(* CODESYS project A2HTC_VISU.project

Project tree, tasks and I/O mapping:
  Device : 750-8212 PFC200, WAGO, order no. 750-8212, version 6.3.0.12
    application Application
      libraries: Standard, 3.5.18.0 (System); CmpBitmapPool, * (System); VisuDialogs, * (System); Util, 3.5.21.0 (System); WagoSysModule_75x_640, 1.9.1.0 (WAGO); WagoAppTime, 1.7.3.5 (WAGO); SysTypes, * (System); SysTime, 3.5.17.0 (System); SysTimeRtc, * (System); CmpLog, * (System); CommFB, * (3S - Smart Software Solutions GmbH)
      task VISU_TASK (cyclic, interval 100 ms, priority 15) calls VisuElems.Visu_Prg, VisuSync
      task TrendRecordingTask (cyclic, interval 100 ms, priority 15) calls VisuTrendStorageAccess.GlobalInstances.g_TrendRecordingManager.CyclicCall
      task MainTask (cyclic, interval 200 ms, priority 15) calls PLC_PRG, readtest, TrendStorageAPI_TestProg
      visualisation Page
      Prog/
        function FctSetDefaultDataCurve [ST]
        program Prog [ST]
      visualisation Visualization_1
      text list TextList
      Trend Recording Manager
        Visualization_1_Trend1
        Visualization_1_Trend2
        Trend1
        Visualization_1_Trend3
      Overlap/
        function FctGetXYValues [ST]
        data type ENUM_CMD_PENDING
        program Overlap [ST]
      program PLC_PRG [ST]
      data type STATUS
      visualisation Visualization
      program VisuSync [ST]
      data type LIMITS
      visualisation Visualization_2
      function block VISU [ST]
      function LIMIT_CHECK [ST]
      data type UNIT
      image pool ImagePool
      global variables GVL
      data type GRAPH_AXIS
      function block READ_TRENDS [ST]
      function block FB_TrendConsumer [ST]: SetDestination, ErrorOccurred, ReadingDataCompleted, TimestampRead, ValueRead, VariableConfigurationRead
      function block FB_ReadTrend [ST]
      function DAY_TO_TIME [ST]
      function block CYCLE_TIME [ST]
      function T_PLC_MS [ST]
      program readtest [ST]
      program TrendStorageAPI_TestProg [ST]
      function block TrendStorageReaderConsumer [ST]: VariableConfigurationRead, ErrorOccurred, TimestampRead, ValueRead, ReadingDataCompleted, SetDestination
      function block TrendStorageWriterListener [ST]: DataWritten
      Visualizations/
        visualisation MinMaxTimestamps
        visualisation ReadValues
        visualisation NewDataWritten
    Kbus : Kbus, WAGO, version 2.1.0.1
        unmapped channels: K-BUS diagnostics
    Serial
      COM1 : COM1, WAGO, version 0.0.0.19
  libraries: VisuSymbols, 4.5.0.0 (System); WagoVisuIcons, 1.1.0.8 (WAGO); WagoVisuIconsMaterialDesign, 1.0.0.2 (WAGO)
  5ce3da45-db07-42e7-a21c-a00fff4ed8f6|C:\Users\MartinStark\Documents\A2HTC\VISU\Grün\Temp_Hum_OK.svg
  5ce3da45-db07-42e7-a21c-a00fff4ed8f6|C:\Users\MartinStark\Documents\A2HTC\VISU\Grün\Cooling_OK.svg
  5ce3da45-db07-42e7-a21c-a00fff4ed8f6|C:\Users\MartinStark\Documents\A2HTC\VISU\Rot\FAN_ERROR.svg
  5ce3da45-db07-42e7-a21c-a00fff4ed8f6|C:\Users\MartinStark\Documents\A2HTC\VISU\Gelb\Hum_WARN.svg
  5ce3da45-db07-42e7-a21c-a00fff4ed8f6|C:\Users\MartinStark\Documents\A2HTC\VISU\Rot\Heating_ERROR.svg
  5ce3da45-db07-42e7-a21c-a00fff4ed8f6|C:\Users\MartinStark\Documents\A2HTC\VISU\Grün\Heating_OK.svg
  5ce3da45-db07-42e7-a21c-a00fff4ed8f6|C:\Users\MartinStark\Documents\A2HTC\VISU\Gelb\Heating_WARN.svg
  5ce3da45-db07-42e7-a21c-a00fff4ed8f6|C:\Users\MartinStark\Documents\A2HTC\VISU\Gelb\FAN_WARN.svg
  5ce3da45-db07-42e7-a21c-a00fff4ed8f6|C:\Users\MartinStark\Documents\A2HTC\VISU\Gelb\Cooling_WARN.svg
  5ce3da45-db07-42e7-a21c-a00fff4ed8f6|C:\Users\MartinStark\Documents\A2HTC\VISU\Grün\FAN_OK.svg
  text list GlobalTextList
  5ce3da45-db07-42e7-a21c-a00fff4ed8f6|C:\Users\MartinStark\Documents\A2HTC\VISU\Rot\Cooling_ERROR.svg
  5ce3da45-db07-42e7-a21c-a00fff4ed8f6|C:\Users\MartinStark\Documents\A2HTC\VISU\Gelb\Temp_Hum_WARN.svg
  5ce3da45-db07-42e7-a21c-a00fff4ed8f6|C:\Users\MartinStark\Documents\A2HTC\VISU\Hintergrund.png
  5ce3da45-db07-42e7-a21c-a00fff4ed8f6|C:\Users\MartinStark\Documents\A2HTC\VISU\Rot\Temp_Hum_ERROR.svg
  5ce3da45-db07-42e7-a21c-a00fff4ed8f6|C:\Users\MartinStark\Documents\A2HTC\VISU\Rot\Hum_ERROR.svg
  5ce3da45-db07-42e7-a21c-a00fff4ed8f6|C:\Users\MartinStark\Documents\A2HTC\VISU\A2HTC.png
  5ce3da45-db07-42e7-a21c-a00fff4ed8f6|C:\Users\MartinStark\Documents\A2HTC\VISU\Grün\HUM_OK.svg
  5ce3da45-db07-42e7-a21c-a00fff4ed8f6|C:\Users\MartinStark\Documents\GitHub\PLS\Mirroring_Webvisu\graph\visu\Model_Viewer\model\Image_0.png
  5ce3da45-db07-42e7-a21c-a00fff4ed8f6|C:\Users\MartinStark\Documents\GitHub\PLS\Mirroring_Webvisu\graph\visu\Model_Viewer\model\Fox.bin
  5ce3da45-db07-42e7-a21c-a00fff4ed8f6|C:\Users\MartinStark\Documents\GitHub\PLS\Mirroring_Webvisu\graph\visu\Model_Viewer\model\Fox.gltf
  5ce3da45-db07-42e7-a21c-a00fff4ed8f6|C:\Users\MartinStark\Documents\GitHub\PLS\Mirroring_Webvisu\graph\visu\Model_Viewer\model\AlloySand2_bump_normalmap.png
  5ce3da45-db07-42e7-a21c-a00fff4ed8f6|C:\Users\MartinStark\Documents\GitHub\PLS\Mirroring_Webvisu\graph\visu\Model_Viewer\model\I5C3D083F677C41699172E93241A6F1D3basecolortexture.png
  5ce3da45-db07-42e7-a21c-a00fff4ed8f6|C:\Users\MartinStark\Documents\GitHub\PLS\Mirroring_Webvisu\graph\visu\Model_Viewer\model\ICA6ACE20800D44CEA1C27E63EFB994CEbasecolortexture.png
  5ce3da45-db07-42e7-a21c-a00fff4ed8f6|C:\Users\MartinStark\Documents\GitHub\PLS\Mirroring_Webvisu\graph\visu\Model_Viewer\model\MetalsOrnamentalMetalsAluminumBrushed_normalmap.png
  5ce3da45-db07-42e7-a21c-a00fff4ed8f6|C:\Users\MartinStark\Documents\A2HTC\VISU\Schriftarten Test\Bahnschrift Light.svg
  5ce3da45-db07-42e7-a21c-a00fff4ed8f6|C:\Users\MartinStark\Documents\A2HTC\VISU\Schriftarten Test\ISOCPEUR.svg
  5ce3da45-db07-42e7-a21c-a00fff4ed8f6|C:\Users\MartinStark\Documents\A2HTC\VISU\Schriftarten Test\Segoe UI Light.svg
  5ce3da45-db07-42e7-a21c-a00fff4ed8f6|C:\Users\MartinStark\Documents\A2HTC\VISU\Schriftarten Test\Yu Gothic UI Light.svg
  5ce3da45-db07-42e7-a21c-a00fff4ed8f6|C:\Users\MartinStark\Documents\A2HTC\VISU\Schriftarten Test\Arial Nova Light.svg
*)

// Device/Application/STATUS
TYPE STATUS :
STRUCT
	OK      : BOOL;
	WARNING : BOOL;
	ERROR   : BOOL;
END_STRUCT
END_TYPE

// Device/Application/LIMITS
TYPE LIMITS :
STRUCT
	UPPER_LIMIT : REAL := 25;
	LOWER_LIMIT : REAL := 22.5;
END_STRUCT
END_TYPE

// Device/Application/Overlap/ENUM_CMD_PENDING
{attribute 'qualified_only'}
{attribute 'strict'}
TYPE ENUM_CMD_PENDING :
(
	NO_CMD,         // no command pending
	UPDATE,         // Update pending
	CLEAN           // Clean pending
);
END_TYPE

// Device/Application/UNIT
TYPE UNIT :
STRUCT
	VALUE   : REAL := 23.5;
	STATUS  : STATUS;
	LIMITS  : LIMITS;
END_STRUCT
END_TYPE

// Device/Application/GRAPH_AXIS
TYPE GRAPH_AXIS :
STRUCT
	sLabel: STRING;
	aData: ARRAY[0..1000] OF REAL;
    diNumOfData : DINT;
	sBorderColor : STRING;
	xFill : BOOL;
END_STRUCT
END_TYPE

// Device/Application/GVL
{attribute 'qualified_only'}
VAR_GLOBAL
	TEMP_DEV_STATUS       : DWORD;
	HUM_DEV_STATUS        : DWORD;
	FAN_DEVICE_STATUS     : DWORD;
	HEATING_DEVICE_STATUS : DWORD;
	COOLING_DEVICE_STATUS : DWORD;
	
	TEMP       : UNIT;
	TEMP_LIMIT : LIMITS;
	HUM        : UNIT;
	HUM_LIMIT  :LIMITS;
	AIRFLOW    : UNIT;
	FAN        : UNIT;
	HEAT       : UNIT;
	COOLING    : UNIT;
	
	AIRFLOW_LIMIT : LIMITS;
	HEAT_POWER : REAL;
	COOL_POWER : REAL;
	just_true : BOOL := TRUE;
END_VAR

// Device/Application/VisuSync
PROGRAM VisuSync

VAR_INPUT
   udiCycleCounter : UDINT;
END_VAR

udiCycleCounter := udiCycleCounter +1;

END_PROGRAM

// Device/Application/PLC_PRG
PROGRAM PLC_PRG
VAR
	generator1 : GEN;
	iSignal1 : INT;
	rSignalToRecord1 : REAL;
	xRecord : BOOL;
	random_temp : REAL;
	random_hum  : REAL;
	always_true : BOOL:= TRUE;
    (* Define the struct variable *)
    myAxis : GRAPH_AXIS;
    
    (* Trigger variable to update data *)
    bUpdateChart : BOOL := FALSE;
    
    sInputLabels : STRING(1000); 
	
	first_cycle : BOOL:= FALSE;
	
	
	
	
	
	
	
    (* Function Block Instance *)
    fbTrendReader : FB_ReadTrend;
    
    (* Data Structure for the Chart *)
    stMyChartData : GRAPH_AXIS;
    sMyLabels : STRING(2000);
    
    (* Control Variables *)
    xReadTrigger : BOOL;
    xDone : BOOL;
    xBusy : BOOL;
    xError : BOOL;
    sErrorMessage : STRING;
    
    (* Parameters *)
    dtStartTime : DT;
    dtEndTime : DT;
    sTrendName : STRING := 'Trend1'; (* MUST match the Trend Recording name in Visualization Manager *)
    
    (* Helper to calc times *)
    tDuration : TIME := T#1H; (* Read last 1 hour *)
    // fbGetTime : GetLocalTime; (* Placeholder: Use system specific time FB *)
    dtNow : DT := DT#2024-01-01-10:00:00; 
    
	
	
    stChartData : GRAPH_AXIS;
    xInit : BOOL := TRUE;	
	
	fbCycleTime : CYCLE_TIME;
	
	
    dtNow2 : DT;
    sCurrentTime : STRING;
	
	

    Result : RTS_IEC_RESULT;

    ltodNow : LTIME_OF_DAY;
    ldatNow : LDATE;
	
    stUTC_DateAndTime : SysTimeRtc.SYSTIME;
    ldtNow : LDATE_AND_TIME;
    udiResult : RTS_IEC_RESULT;
	
	
	
	
END_VAR











IF random_temp > 40 THEN
	random_temp := 0;
ELSE 
	random_temp := random_temp + 2;
END_IF

IF random_hum > 80 THEN
	random_hum := 0;
ELSE 
	random_hum := random_hum + 1;
END_IF



generator1(MODE := GEN_MODE.SINE, BASE := TRUE, PERIOD := TIME#10S, AMPLITUDE := 500, OUT => iSignal1);
rSignalToRecord1 := INT_TO_REAL(iSignal1)/100 + 20; 
xRecord := rSignalToRecord1 >= 20;




(* Initialize only once or on demand *)
IF xInit THEN
    (* 1. Set Style Properties - Using fields from graph/db/GRAPH_AXIS.ST *)
    stChartData.sLabel := 'Fixed Values Demo';
    stChartData.sBorderColor := 'rgb(54, 162, 235)'; (* Blue *)
    stChartData.xFill := FALSE;

    (* 2. Set 10 Fixed Data Points *)
    stChartData.aData[0] := 10.0;
    stChartData.aData[1] := 20.0;
    stChartData.aData[2] := 15.5;
    stChartData.aData[3] := 25.0;
    stChartData.aData[4] := 30.0;
    stChartData.aData[5] := 10.0;
    stChartData.aData[6] := 5.0;
    stChartData.aData[7] := 12.0;
    stChartData.aData[8] := 18.0;
    stChartData.aData[9] := 22.0;
    
    (* Set the number of valid data points *)
    stChartData.diNumOfData := 10;
       
    xInit := FALSE;
END_IF

END_PROGRAM

// Device/Application/FB_ReadTrend
FUNCTION_BLOCK FB_ReadTrend
VAR_INPUT
	xExecute : BOOL;
    sTrendName : STRING; 
    tStartTime : DT;
    tEndTime : DT;
    iChannelIndex : INT := 0; 
END_VAR
VAR_OUTPUT
	sLabels : STRING(2000); 
    xDone : BOOL;
    xBusy : BOOL;
    xError : BOOL;
    sError : STRING;
END_VAR
VAR
	step : INT := 0;
    fbTrendReader : VisuTrendStorageAccess.TrendStorageReader;
    fbTrendConsumer : FB_TrendConsumer;
    
    liStart : LINT;
    liEnd : LINT;
    eResult : VisuTrendStorageAccess.ETrendStorageReaderErrors;
END_VAR
VAR_IN_OUT
    stChartData : GRAPH_AXIS;
END_VAR


CASE step OF
    0: (* Idle *)
        IF xExecute THEN
            xBusy := TRUE;
            xDone := FALSE;
            xError := FALSE;
            sError := '';
            
            // Set up Consumer
            fbTrendConsumer.SetDestination(ADR(stChartData), ADR(sLabels), tStartTime);
            
            // Initialize Reader
            fbTrendReader.Initialize(sTrendName); // User docu says Initialize exists. Assuming sTrendName arg.
            
            // Convert DT to LINT (Timestamp). DT is seconds. Trend usually ms.
            liStart := DT_TO_LINT(tStartTime) * 1000;
            liEnd := DT_TO_LINT(tEndTime) * 1000;
            
            step := 10;
        END_IF
        
    10: (* Start Read *)
        eResult := fbTrendReader.Read(
            liTimstampFrom := liStart,
            liTimstampTo := liEnd,
            itfTrendStorageReaderConsumer := fbTrendConsumer
        );
        
        IF eResult = VisuTrendStorageAccess.ETrendStorageReaderErrors.NoError THEN
             // Done immediately (unlikely for large data but possible)
             stChartData.sLabel := 'Trend Data';
             stChartData.sBorderColor := 'blue';
             stChartData.xFill := FALSE;
             step := 20;
        ELSIF eResult = VisuTrendStorageAccess.ETrendStorageReaderErrors.AdditionalReadCallRequired THEN
             step := 11; // Continue Reading
        ELSIF eResult = VisuTrendStorageAccess.ETrendStorageReaderErrors.NotInitialized THEN
             sError := 'Not Initialized';
             xError := TRUE;
             step := 99;
        ELSE
             sError := 'Read Error';
             xError := TRUE;
             step := 99;
        END_IF
        
    11: (* Continue Reading *)
        eResult := fbTrendReader.ContinueReading(
            liTimstampFrom := liStart,
            liTimstampTo := liEnd,
            itfTrendStorageReaderConsumer := fbTrendConsumer
        );

         IF eResult = VisuTrendStorageAccess.ETrendStorageReaderErrors.NoError THEN
             step := 20;
         ELSIF eResult = VisuTrendStorageAccess.ETrendStorageReaderErrors.AdditionalReadCallRequired THEN
             // Stay in step 11
         ELSE
             sError := 'Continue Error';
             xError := TRUE;
             step := 99;
         END_IF

    20: (* Done *)
        xDone := TRUE;
        xBusy := FALSE;
        IF NOT xExecute THEN
            step := 0;
        END_IF
        
    99: (* Error *)
        xBusy := FALSE;
        IF NOT xExecute THEN
            step := 0;
        END_IF
        
END_CASE

END_FUNCTION_BLOCK

// Device/Application/FB_TrendConsumer
FUNCTION_BLOCK FB_TrendConsumer IMPLEMENTS VisuTrendStorageAccess.ITrendStorageReaderConsumer
VAR_INPUT
	pChartData : POINTER TO GRAPH_AXIS;
    pLabelString : POINTER TO STRING(2000);
    tStart : DT;
END_VAR
VAR_OUTPUT
END_VAR
VAR
    pAxis : POINTER TO GRAPH_AXIS;
    pLabels : POINTER TO STRING(2000);
    sLabels : STRING(2000); // Internal build buffer
    iMaxLabels : INT := 20;
    tStartTime : DT;
    iCurrentRow : DINT;
    rCurrentVal : REAL;
    xFirst : BOOL := TRUE;
	
    // DEBUG
    debug_CountValueRead : DINT;
    debug_LastLiValue : LINT;
    debug_LastTimestamp : LINT;
    debug_CountTimestampRead : DINT;
    debug_LastTimestampIndex : DINT;
    
    pLReal : POINTER TO LREAL;
END_VAR

METHOD SetDestination
VAR_INPUT
	pChartData : POINTER TO GRAPH_AXIS;
    pLabelString : POINTER TO STRING(2000);
    tStart : DT;
END_VAR
    pAxis := pChartData;
    pLabels := pLabelString;
    tStartTime := tStart;
    
    // Reset
    IF pAxis <> 0 THEN
        pAxis^.diNumOfData := 0;
    END_IF
    IF pLabels <> 0 THEN
        pLabels^ := '[';
        sLabels := '[';
    END_IF
    xFirst := TRUE;
END_METHOD

(* Notification, that an error occurred.*)
METHOD ErrorOccurred
VAR_INPUT
	(* The error, that occurred*)
	eETrendStorageReaderErrors	: VisuTrendStorageAccess.ETrendStorageReaderErrors;
	(* Identifies the step, where the error occurred	*)
	eDuringWhichStep	: VisuTrendStorageAccess.ETrendStorageReaderStep;
END_VAR
END_METHOD

(* Notification, that reading the data (i.e. the values) has been completed.*)
METHOD ReadingDataCompleted
// Finalize labels
IF pLabels <> 0 THEN
	pLabels^ := CONCAT(pLabels^, ']');
END_IF
END_METHOD

(* Notification, that a timestamp from TblTrendData has been read and can be processed.*)
METHOD TimestampRead
VAR_INPUT
	(* A 0-based index of the row read from TblTrendData*)
	diWhichRow	: DINT;
	(* The absolute timestamp, that was read from TblTrendData*)
	liTimestamp	: LINT;


END_VAR
VAR
    sTempLabel : STRING(80);
    ldtCurrent : LDATE_AND_TIME;
    diIndex : DINT;
END_VAR
    // Convert timestamp (uS or mS? Usually uS or mS from Trend. LINT is usually ms or us)
    // Assuming MS since 1970? Or LTIME?
    // Standard Trend timestamps are µs (microseconds) usually.
    // DT is Seconds.
    
    // For label generation:
    // For label generation:
    IF pAxis <> 0 AND pLabels <> 0 THEN
        diIndex := pAxis^.diNumOfData; 
        
        // DEBUG
        debug_CountTimestampRead := debug_CountTimestampRead + 1;
        debug_LastTimestampIndex := diIndex; // Check what index TimestampRead sees
        
        IF diIndex < 100 AND (diIndex < iMaxLabels) THEN
             // ... logic ...
             
             // Convert to LDT (High Res) if liTimestamp is in ms (matches current_time logic)
             // current_time uses: TO_LDT(val * LTIME#1ms)
             ldtCurrent := TO_LDT(liTimestamp * LTIME#1ms);
             
             sTempLabel := LDT_TO_STRING(ldtCurrent);
             // Format: LDT#2025-02-07-13:15:15.369...
             // Take right 15 chars to get "15:15.369..." approx
             sTempLabel := RIGHT(sTempLabel, 15); 
             
             IF NOT xFirst THEN
                 pLabels^ := CONCAT(pLabels^, ', "');
             ELSE
                 pLabels^ := CONCAT(pLabels^, '"');
                 xFirst := FALSE;
             END_IF
             pLabels^ := CONCAT(pLabels^, sTempLabel);
             pLabels^ := CONCAT(pLabels^, '"');
        END_IF
    END_IF
END_METHOD

(* Notification, that a variable value from TblTrendData has been read and can be processed.*)
METHOD ValueRead
VAR_INPUT
	(* A 0-based index of the row read from TblTrendData.*)
	diWhichRow	: DINT;
	(* A 0-based index of the variable within all variables*)
	iWhichVariable	: INT;
	(* The value, that was read from TblTrendData*)
	liValue	: LINT;
	(* Indicates, whether NULL is stored in the trend storage*)
	xValueNULL	: BOOL;
END_VAR
VAR
    diIndex : DINT;
END_VAR
IF pAxis <> 0 THEN
	diIndex := pAxis^.diNumOfData;
	
	debug_CountValueRead := debug_CountValueRead + 1;
	debug_LastLiValue := liValue;
	
	IF diIndex <= 1000 THEN
		 // Debug: check raw value.
		 IF NOT xValueNULL THEN
			// Interpreting bits: liValue (LINT) holds the bits of LREAL (usually).
			// Or REAL? Standard Codesys Trend uses LREAL.
			// We point an LREAL pointer to the address of liValue to read it as float.
			// Then cast to REAL for the chart array.
			pLReal := ADR(liValue);
			pAxis^.aData[diIndex] := TO_REAL(pLReal^); 
		 ELSE
			pAxis^.aData[diIndex] := -9999.0; // Debug nulls
		 END_IF
		 
		 pAxis^.diNumOfData := pAxis^.diNumOfData + 1;
	END_IF
END_IF
END_METHOD

(* Notification, that the variable configuration was read and reading of data will start immediately.*)
METHOD VariableConfigurationRead
VAR_INPUT
	(* Points to an array of TrendStorageVariableDescription Variables,
 where the configuration of the variables has been stored. This array
 contains the description of the variables, whose data will be read*)
	paTrendStorageVariableDescription	: POINTER TO ARRAY [0..0] OF VisuTrendStorageAccess.TrendStorageVariableDescription;
	(* The effective size of the array above, i.e. the number of variables*)
	iCountVariables	: INT;
END_VAR
END_METHOD

END_FUNCTION_BLOCK

// Device/Application/CYCLE_TIME
FUNCTION_BLOCK CYCLE_TIME
VAR_INPUT
	RST : BOOL;
END_VAR
VAR_OUTPUT
	ct_min : TIME;
	ct_max : TIME;
	ct_last : TIME;
	systime : TIME;
	sysdays : INT;
	cycles : DWORD;
END_VAR
VAR
	last_cycle : TIME;
	tx: TIME;
	init: BOOL;
END_VAR


tx := DWORD_TO_TIME(T_PLC_MS()) - last_cycle;
IF rst THEN
	ct_min := t#10h;
	ct_max := t#0ms;
	cycles := 0;
ELSIF last_cycle > t#0s THEN
	IF tx < ct_min THEN ct_min := tx;
	ELSIF tx > ct_max THEN ct_max := tx;
	END_IF;
	ct_last := tx;
ELSIF ct_min = t#0s THEN
	ct_min := t#0s - t#1ms;
END_IF;
IF init THEN
	systime := systime + tx;
		IF systime >= t#1d THEN
			systime := systime - t#1d;
			sysdays := sysdays + 1;
		END_IF;
END_IF;
init := TRUE;
last_cycle := last_cycle + tx;
cycles := cycles + 1;

END_FUNCTION_BLOCK

// Device/Application/T_PLC_MS
FUNCTION T_PLC_MS : DWORD
VAR CONSTANT
	debug : BOOL := 0;
	N : INT := 0;
	offset : DWORD := 0;
END_VAR
VAR
	tx : TIME;
END_VAR


tx := TIME();
T_PLC_MS := TIME_TO_DWORD(Tx);

IF debug THEN
	T_PLC_MS := (SHL(T_PLC_MS,N) OR SHL(DWORD#1,N)-1) + OFFSET;
END_IF;

END_FUNCTION

// Device/Application/readtest
PROGRAM readtest
VAR
	i : INT;
	
	diVal2 : DINT := 1000;
	siVal3 : SINT;
	
	rVal	: REAL;
	rSin	: REAL;
END_VAR

// This program simulates the data, that is written to the trend storage

i := (i + 1) MOD 23;
siVal3 := siVal3 + 1;

IF siVal3 > 0 THEN
	diVal2 := diVal2 + 2;
	
	IF diVal2 > 1100 THEN
		diVal2 := 1000;
	END_IF
END_IF

rVal := rVal +0.05;
rSin := 5 * SIN(rVal);

END_PROGRAM

// Device/Application/TrendStorageAPI_TestProg
// Example program, that access the trend storage
PROGRAM TrendStorageAPI_TestProg
VAR
	xInitialized : BOOL;
	instTrendStorageReader 			: TrendStorageReader; 
	instTrendStorageWriterListener	: TrendStorageWriterListener;
	instTrendStorageReaderConsumer	: TrendStorageReaderConsumer;
	
	// Usecase 1:
	eError							: VisuTrendStorageAccess.ETrendStorageReaderErrors;
	liMinTimestamp					: LINT;
	liMaxTimestamp					: LINT;
	timeDateMin						: SYSTIMEDATE;
	uiMicrosecondsMin				: UINT;
	timeDateMax						: SYSTIMEDATE;
	uiMicrosecondsMax				: UINT;
	
	// Usecase 2:
	xDoReadTest2					: BOOL;
	eError2							: VisuTrendStorageAccess.ETrendStorageReaderErrors;
	liTimstampFrom2					: LINT;
	liTimstampTo2					: LINT;
	iLoopCounter					: INT;
	
	xStopContinueReading			: BOOL;

	xComputeTimestamps				: BOOL;
	xComputeDateTime				: BOOL;
	timeDateFrom2					: SYSTIMEDATE;
	uiMicrosecondsFrom2				: UINT;
	timeDateTo2						: SYSTIMEDATE;
	uiMicrosecondsTo2				: UINT;
	
	
	ChartOne : GRAPH_AXIS;
	sLabelOne : STRING(2000);
	
	    stUTC_DateAndTime : SYSTIME;

    Result : RTS_IEC_RESULT;

    ldtNow : LDATE_AND_TIME;
    ltodNow : LTIME_OF_DAY;
    ldatNow : LDATE;

    stUTC_Timestamp : SysTime;
    stLocal_TimeStamp : SysTime;
    stdNow : SysTimeDate;

    dtNow : DATE_AND_TIME;
    todNow : TIME_OF_DAY;
    datNow : DATE;   
    datToday : DATE; 	
END_VAR

// Required call to Initialize before any methods of the TrendStorageReader instance can be used
Result := SysTimeRtcHighResGet(stUTC_DateAndTime); // UlINT#1738934115369

ldtNow := TO_LDT(stUTC_DateAndTime * LTIME#1ms); // LDT#2025-2-7-13:15:15.369000000
ltodNow := TO_LTOD(ldtNow); // LTOD#13:15:15.369000000
ldatNow := TO_LDATE(ldtNow); // LD#2025-2-7


Result := SysTimeRtcHighResGet(stUTC_Timestamp); // ULINT#1528273494913
Result := SysTimeRtcConvertHighResToLocal(stUTC_Timestamp, stdNow);

Result := SysTimeRtcConvertDateToHighRes(stdNow, stLocal_TimeStamp); // ULINT#1528280694913

dtNow := TO_DT(stLocal_TimeStamp / 1000); // DT#2018-6-6-10:24:54
todNow := TO_TOD(stLocal_TimeStamp MOD TO_ULINT(T#1D)); // TOD#10:24:54.913
datToday := TO_DATE(dtNow); // D#2018-6-6


// Required call to Initialize before any methods of the TrendStorageReader instance can be used
IF NOT xInitialized THEN
	xInitialized := TRUE;
	instTrendStorageReader.Initialize(sPacketName := 'Trend1');
	// Usecase 3: Notification, if new data is available in the trend storage.
	// This optional call is necessary, if we want to be informed, if new data has been written
	// to the trend storage.
	instTrendStorageReader.AddTrendStorageWriterListener(instTrendStorageWriterListener);
END_IF

// Usecase 1: Determine the min/max timestamp range, for which data is available in the trend storage
eError := instTrendStorageReader.GetMinMaxTimestamps(
	liMinTimestamp			=> liMinTimestamp,
	liMaxTimestamp			=> liMaxTimestamp
);

// Comvert the timestamps in a human readable form
TrendStorageConvertFromTimestamp(liTimestamp := liMinTimestamp, timeDate => timeDateMin, uiMicroseconds => uiMicrosecondsMin);
TrendStorageConvertFromTimestamp(liTimestamp := liMaxTimestamp, timeDate => timeDateMax, uiMicroseconds => uiMicrosecondsMax);

// Usecase 2: Read values from the trend storage
// The data returned by the read process is truncated into small pieces. The 1st call is a call
// of method Read. In case of return code VisuTrendStorageAccess.ETrendStorageReaderErrors.AdditionalReadCallRequired
// additional calls are necessary, but calls to method ContinueReading.
IF eError2 = VisuTrendStorageAccess.ETrendStorageReaderErrors.AdditionalReadCallRequired THEN
	iLoopCounter := iLoopCounter + 1;
	VisuElems.Visu_Output_2('Call to ContinueReading ', INT_TO_STRING(iLoopCounter), 4);
	eError2 := instTrendStorageReader.ContinueReading(
		liTimstampFrom					:= liTimstampFrom2,
		liTimstampTo					:= liTimstampTo2,
		itfTrendStorageReaderConsumer	:= instTrendStorageReaderConsumer
	);
END_IF

IF xDoReadTest2 THEN
	xDoReadTest2 := FALSE;

	iLoopCounter := 0;
	instTrendStorageReaderConsumer.diTotalCountRows := 0;
	
	instTrendStorageReaderConsumer.SetDestination(pChartData := ADR(ChartOne), pLabelString := ADR(sLabelOne), tStart := dtNow);

	// Always read full range
    liTimstampFrom2 := liMinTimestamp;
    liTimstampTo2 := liMaxTimestamp;
	
	eError2 := instTrendStorageReader.Read(
		liTimstampFrom					:= liTimstampFrom2,
		liTimstampTo					:= liTimstampTo2,
		itfTrendStorageReaderConsumer	:= instTrendStorageReaderConsumer
	);
END_IF

// This helps us to abort a long running read call
IF xStopContinueReading THEN
	xStopContinueReading := FALSE;
	// This stops the reading
	eError2 := VisuTrendStorageAccess.ETrendStorageReaderErrors.NoError;
END_IF

IF xComputeTimestamps THEN
	xComputeTimestamps := FALSE;
	
	liTimstampFrom2 := TrendStorageConvertToTimestamp(timeDateFrom2, uiMicrosecondsFrom2);
	liTimstampTo2 := TrendStorageConvertToTimestamp(timeDateTo2, uiMicrosecondsTo2);
END_IF

IF xComputeDateTime THEN
	 xComputeDateTime := FALSE;
	 
	TrendStorageConvertFromTimestamp(liTimestamp := liTimstampFrom2, timeDate => timeDateFrom2, uiMicroseconds => uiMicrosecondsFrom2);
	TrendStorageConvertFromTimestamp(liTimestamp := liTimstampTo2, timeDate => timeDateTo2, uiMicroseconds => uiMicrosecondsTo2);
END_IF

END_PROGRAM

// Device/Application/TrendStorageWriterListener
// Example function block, that will be informed, if new data has been written to the
// trend storage. It simply stores the information, that is displayed in the visualization
// "ReadValues"
FUNCTION_BLOCK TrendStorageWriterListener IMPLEMENTS ITrendStorageWriterListener
VAR
	m_liFirstTimestamp	: LINT;
	m_liLastTimestamp	: LINT;
	m_iCountRows		: INT;
	
	m_timeDateMin		: SYSTIMEDATE;
	m_uiMicrosecondsMin	: UINT;
	m_timeDateMax		: SYSTIMEDATE;
	m_uiMicrosecondsMax	: UINT;
END_VAR

(* Notification, that data has been written to the trend storage*)
METHOD DataWritten
VAR_INPUT
	(* The first timestamp for which data was written to the trend storage*)
	liFirstTimestamp	: LINT;
	(* The last timestamp for which data was written to the trend storage*)
	liLastTimestamp	: LINT;
	(* The number of rows, that have been written to the trend storage*)
	iCountRows	: INT;
END_VAR
m_liFirstTimestamp := liFirstTimestamp;
m_liLastTimestamp := liLastTimestamp;
m_iCountRows := iCountRows;

// Comvert the timestamps in a human readable form
TrendStorageConvertFromTimestamp(liTimestamp := liFirstTimestamp, timeDate => m_timeDateMin, uiMicroseconds => m_uiMicrosecondsMin);
TrendStorageConvertFromTimestamp(liTimestamp := liLastTimestamp, timeDate => m_timeDateMax, uiMicroseconds => m_uiMicrosecondsMax);
END_METHOD

END_FUNCTION_BLOCK

// Device/Application/TrendStorageReaderConsumer
// This function block is a simple example implementation of the ITrendStorageReaderConsumer interface.
FUNCTION_BLOCK TrendStorageReaderConsumer IMPLEMENTS ITrendStorageReaderConsumer
VAR_INPUT
	// If this flag is TRUE an output like a csv export will be generated. Should be only
	// used, if not too much data is read from the trend storage
	xDetailedOutput						: BOOL;
	
	// This member is used to track the total number of rows, that have been read from the trend storage
	diTotalCountRows					: DINT;
END_VAR
VAR
	// This instance converts the values into a suitable representation, e.g. into a string
	m_instValueConverter				: TrendStorageReaderValueConverter;	

	// A line used to collect the data read from the trend storage
	m_sLine								: STRING(255);
	// Used to identify the rows
	m_diWhichRow						: DINT;
	
	m_diRowCounter						: DINT;
	// Used to track the minimum/maximum timestamp, that was read
	m_liTimestampMin					: LINT := 16#1FFFFFFFFFFFFFFF;
	m_liTimestampMax					: LINT := 0;
	
	
	pAxis : POINTER TO GRAPH_AXIS;
    pLabels : POINTER TO STRING(2000);
    sLabels : STRING(2000);
    tStartTime : DT;
    xFirst : BOOL;	
	

    
    rLastNonZeroValue : REAL;	
	
    // Deep Debugging
    liLastRawValue : LINT;
    iLastVarIndex : INT;
    diValueReadCalls : DINT;
    xLastNull : BOOL;	
END_VAR

METHOD VariableConfigurationRead
VAR_INPUT
	paTrendStorageVariableDescription	: POINTER TO ARRAY [0..0] OF VISUTRENDSTORAGEACCESS.TrendStorageVariableDescription;
	iCountVariables	: INT;
END_VAR
m_instValueConverter.SetVariableConfiguration(paTrendStorageVariableDescription, iCountVariables);

// If we previously collected data, we dump it
//ReadingDataCompleted();

VisuElems.Visu_Output_3('New configuration having ', INT_TO_STRING(iCountVariables), ' variables', 4);
END_METHOD

METHOD ErrorOccurred
VAR_INPUT
	(* The error, that occurred*)
	eETrendStorageReaderErrors	: VISUTRENDSTORAGEACCESS.ETrendStorageReaderErrors;
	(* Identifies the step, where the error occurred	*)
	eDuringWhichStep	: VISUTRENDSTORAGEACCESS.ETrendStorageReaderStep;
END_VAR
// Error processing can be done here...
END_METHOD

(* Notification, that a timestamp from TblTrendData has been read and can be processed.*)
METHOD TimestampRead
VAR_INPUT
	(* A 0-based index of the row read from TblTrendData*)
	diWhichRow	: DINT;
	
	(* The absolute timestamp, that was read from TblTrendData*)
	liTimestamp	: LINT;
END_VAR
VAR
	timeDate		: SYSTIMEDATE;
	uiMicroseconds	: UINT;
END_VAR

IF xDetailedOutput THEN
	IF LEN(m_sLine) <> 0 THEN
		VisuElems.Visu_Output_3(DINT_TO_STRING(m_diWhichRow), ': ', m_sLine, 4);
	END_IF
	m_sLine := '';
END_IF

m_diWhichRow := diWhichRow;


IF xDetailedOutput THEN
	// We begin a new line
	m_sLine := LINT_TO_STRING(liTimestamp);

	// Comvert the timestamps in a human readable form
	TrendStorageConvertFromTimestamp(liTimestamp := liTimestamp, timeDate => timeDate, uiMicroseconds => uiMicroseconds);

	// We also append the timestamp in the human readable way
	m_sLine := CONCAT(m_sLine, ';');
	m_sLine := CONCAT(m_sLine, WORD_TO_STRING(timeDate.wYear));
	m_sLine := CONCAT(m_sLine, '-');
	m_sLine := CONCAT(m_sLine, WORD_TO_STRING(timeDate.wMonth));
	m_sLine := CONCAT(m_sLine, '-');
	m_sLine := CONCAT(m_sLine, WORD_TO_STRING(timeDate.wDay));
	m_sLine := CONCAT(m_sLine, ' ');
	m_sLine := CONCAT(m_sLine, WORD_TO_STRING(timeDate.wHour));
	m_sLine := CONCAT(m_sLine, ':');
	m_sLine := CONCAT(m_sLine, WORD_TO_STRING(timeDate.wMinute));
	m_sLine := CONCAT(m_sLine, ':');
	m_sLine := CONCAT(m_sLine, WORD_TO_STRING(timeDate.wSecond));
	m_sLine := CONCAT(m_sLine, ':');
	m_sLine := CONCAT(m_sLine, WORD_TO_STRING(timeDate.wMilliseconds));
	m_sLine := CONCAT(m_sLine, ':');
	m_sLine := CONCAT(m_sLine, UINT_TO_STRING(uiMicroseconds));
ELSE
	m_diRowCounter := m_diRowCounter + 1;
	
	m_liTimestampMax := MAX(m_liTimestampMax, liTimestamp);
	
	(* Append to Label String - Protect against overflow *)
	IF pLabels <> 0 AND LEN(pLabels^) < 1900 THEN
	    TrendStorageConvertFromTimestamp(liTimestamp := liTimestamp, timeDate => timeDate, uiMicroseconds => uiMicroseconds);
	    
	    IF NOT xFirst THEN
	        pLabels^ := CONCAT(pLabels^, ','); // Add comma separator
	    END_IF
	    xFirst := FALSE; 
	    
	    pLabels^ := CONCAT(pLabels^, '"');
	    pLabels^ := CONCAT(pLabels^, WORD_TO_STRING(timeDate.wHour));
	    pLabels^ := CONCAT(pLabels^, ':');
	    pLabels^ := CONCAT(pLabels^, WORD_TO_STRING(timeDate.wMinute));
	    pLabels^ := CONCAT(pLabels^, ':');
	    pLabels^ := CONCAT(pLabels^, WORD_TO_STRING(timeDate.wSecond));
	    pLabels^ := CONCAT(pLabels^, '"');
	END_IF
END_IF
END_METHOD

METHOD ValueRead
VAR_INPUT
	(* A 0-based index of the row read from TblTrendData.*)
	diWhichRow	: DINT;
	(* A 0-based index of the variable within all variables*)
	iWhichVariable	: INT;
	(* The value, that was read from TblTrendData*)
	liValue	: LINT;
	(* Indicates, whether NULL is stored in the trend storage*)
	xValueNULL	: BOOL;
END_VAR
VAR
	sValue		: STRING;
END_VAR

// Debug Capture
diValueReadCalls := diValueReadCalls + 1;
liLastRawValue := liValue;
iLastVarIndex := iWhichVariable;
xLastNull := xValueNULL;

IF xDetailedOutput THEN
	// We simply append the value to the line, that simulates a line of a csv file
	m_sLine := CONCAT(m_sLine, ';');
	
	sValue := m_instValueConverter.ConvertToString(iWhichVariable, liValue, xValueNULL);
	m_sLine := CONCAT(m_sLine, sValue);
ELSE
    IF pAxis <> 0 THEN
        IF iWhichVariable = 0 AND NOT xValueNULL THEN
             IF pAxis^.diNumOfData <= 1000 THEN
                // Use converter to handle potential REAL/INT types correctly via string representation
                sValue := m_instValueConverter.ConvertToString(iWhichVariable, liValue, xValueNULL);
                pAxis^.aData[pAxis^.diNumOfData] := STRING_TO_REAL(sValue);
                
                IF pAxis^.aData[pAxis^.diNumOfData] <> 0 THEN
                    rLastNonZeroValue := pAxis^.aData[pAxis^.diNumOfData];
                END_IF
                
                pAxis^.diNumOfData := pAxis^.diNumOfData + 1;
            END_IF       
        END_IF
    END_IF

END_IF
END_METHOD

{attribute '''DOCU__COMMENT' := ' Notification, that reading the data (i.e. the values) has been completed.'}
(* Notification, that reading the data (i.e. the values) has been completed.*)
METHOD ReadingDataCompleted

VAR
	CMPID_LigLog: UDINT;
	sLogMessage : STRING(255);
END_VAR
IF xDetailedOutput THEN
	IF LEN(m_sLine) <> 0 THEN
		VisuElems.Visu_Output_3(DINT_TO_STRING(m_diWhichRow), ': ', m_sLine, 4);
	END_IF
	m_sLine := '';
ELSE
	diTotalCountRows := diTotalCountRows + m_diRowCounter;

	sLogMessage := CONCAT('ReadingDataCompleted, m_diRowCounter = ', CONCAT('ReadingDataCompleted, m_diRowCounter = ', CONCAT(', diTotalCountRows = ', DINT_TO_STRING(diTotalCountRows))));
	//LogAdd2(LOG_STD_LOGGER, 0, CmpLog.LogClass.LOG_INFO, 0, 0, sLogMessage);
	
	// Prepare for next loops
	m_diRowCounter := 0;
	m_liTimestampMin := 16#1FFFFFFFFFFFFFFF;
	m_liTimestampMax := 0;
	
	
	IF pLabels <> 0 THEN
	    pLabels^ := CONCAT(pLabels^, ']');
	END_IF	
END_IF
END_METHOD

METHOD SetDestination : BOOL
VAR_INPUT
    pChartData : POINTER TO GRAPH_AXIS;
    pLabelString : POINTER TO STRING(2000);
    tStart : DT;
END_VAR
    pAxis := pChartData;
    pLabels := pLabelString;
    tStartTime := tStart;
    
    // Reset
    IF pAxis <> 0 THEN
        pAxis^.diNumOfData := 0;
    END_IF
    IF pLabels <> 0 THEN
        pLabels^ := '[';
        sLabels := '[';
    END_IF
    xFirst := TRUE;
END_METHOD

END_FUNCTION_BLOCK

// Device/Application/Overlap/FctGetXYValues
/// Get X & Y values
FUNCTION FctGetXYValues : bool

VAR_INPUT
   iValue : INT;                     // Input value for calculation  
	rXValue : REFERENCE TO REAL;      // X value 
	rYValue : REFERENCE TO REAL;      // Y value 
END_VAR

VAR
   rValue : REAL;
END_VAR

// X = t − 2 sin t
// Y = 2 − 2 cos t

rValue  := INT_TO_REAL(iValue);
rValue  := rValue/10.0;
rXValue := rValue - 2.0*SIN(rValue);
rYValue := 2.0 - 2.0*COS(rValue);

END_FUNCTION

// Device/Application/Prog/FctSetDefaultDataCurve
/// Set default data for curves
FUNCTION FctSetDefaultDataCurve : bool

VAR
   ix : INT;
END_VAR

// Clean up the arrays
FOR ix := 1 TO 100 BY 1 DO
    Prog.DataX1[ix]  := 0.0 ;
    Prog.DataY1[ix]  := 0.0 ;
END_FOR
   
// Set deualt data   
Prog.DataX1[1] := -10.0 ;
Prog.DataX1[2] := 20.0 ;
Prog.DataX1[3] := 30.0 ;
Prog.DataX1[4] := 40.0 ;
Prog.DataX1[5] := 50.0 ;  
Prog.DataX1[6] := 60.0 ;  
Prog.DataX1[7] := 70.0 ;  
Prog.DataX1[8] := 80.0 ;  
Prog.DataX1[9] := 90.0 ;  
Prog.DataX1[10] := 100.0 ;  

Prog.DataY1[1] := 10.0 ;
Prog.DataY1[2] := 20.0 ;
Prog.DataY1[3] := 10.0 ;
Prog.DataY1[4] := 30.0 ;
Prog.DataY1[5] := 10.0 ;
Prog.DataY1[6] := 40.0 ;
Prog.DataY1[7] := 10.0 ;
Prog.DataY1[8] := 50.0 ;
Prog.DataY1[9] := 10.0 ;
Prog.DataY1[10] := 60.0 ;

END_FUNCTION

// Device/Application/Prog/Prog
PROGRAM Prog

VAR_INPUT
	xyChart: VisuStructXYChart;         // Variable for element configuration
   
	AxisX: VisuStructXYChartAxis;       // Variable for dynamic X axis configuration
	AxisY1 : VisuStructXYChartAxis;     // Variable for dynamic Y1 axis configuration
   
   Curve1 : VisuStructXYChartCurve;    // Variable for dynamic curve 1 configuration

   // Arrays of data used for curves   
   DataX1 : ARRAY [1..100] OF REAL ;
   DataY1 : ARRAY [1..100] OF REAL ;

   iCurve1ProgType : INT;              // How to programm the curve 1, 0=modify existig, 1=create a new one
   xProgCurve1 : BOOL;                 // Start programming curve 1

   xProgOff : BOOL;                    // Stop programming
   xProgSave : BOOL;                   // Save the curve
   xProgUndoS : BOOL;                  // Undo single point   
   xProgUndo : BOOL;                   // Undo all the curve
   xSetOrigCurve : BOOL;               // Set original curves
   
   sProgClient : STRING;               // On which client programming is active
   xProgMode : BOOL;                   // Element is in programming mode   
   xChangePending : BOOL;              // Change is pending
   
   udiCycleCounter : UDINT;
END_VAR

VAR
   xInitDone : BOOL;             // If the initialization has been done correctly

   // Here we save the initial element configuration   
	SVxyChart : VisuStructXYChart;
	SVAxisX   : VisuStructXYChartAxis;
	SVAxisY1  : VisuStructXYChartAxis;
   SVCurve1  : VisuStructXYChartCurve;

   xDoIt            : BOOL;
   xDelayProgCurve1 : BOOL;
   xDelayProgOff    : BOOL;
   xDelayProgSave   : BOOL;
   
   rTrigProgCurve1 :  R_TRIG;    // Trigger to detect start programming curve 1 
   rTrigProgOff    :  R_TRIG;    // Trigger to detect stop programming
   rTrigOrig       :  R_TRIG;    // Trigger to detect set original curves
   rTrigUndoS      :  R_TRIG;    // Trigger to detect undo single point
   rTrigUndo       :  R_TRIG;    // Trigger to detect undo curve
   rTrigSave       :  R_TRIG;    // Trigger to detect save curve
   
   random_temp : REAL;
   random_hum  : REAL;
END_VAR

(**********************************************************************************************
   The scope of this application is to show how to use XYChart element in programming mode.
   It simply shows a predefine curve that the user can modify or completely make from scratch.
***********************************************************************************************)


IF random_temp > 60 THEN
	random_temp := 0;
ELSE 
	random_temp := random_temp + 2;
END_IF

IF random_hum > 80 THEN
	random_hum := 0;
ELSE 
	random_hum := random_hum + 1;
END_IF



//------------------------------------------------------------------
// During the first entry we do some initial activities
IF NOT xInitDone THEN
   IF ABS(VisuSync.udiCycleCounter - udiCycleCounter) > 2 THEN    // Valid when "Visu" is running
      // We save the initial element configuration for further uses
      SVxyChart := xyChart;
      SVAxisX   := AxisX;
      SVAxisY1  := AxisY1;
      SVCurve1  := Curve1;

      // We limit the use of the array
      Curve1.diIndexMin := 1 ;        
      Curve1.diIndexMax := 10 ;
      
      FctSetDefaultDataCurve();  // Set default data for curves   
      
      xInitDone := TRUE;         // done
   ELSE
      RETURN ;                   // We will do nothing if we don't' have the correct data          
	END_IF
END_IF


//------------------------------------------------------------------
// We start the programming on curve 
rTrigProgCurve1(CLK:=xProgCurve1, Q=>xDoIt);
IF xDoIt THEN
   xProgCurve1 := FALSE;
   rTrigProgCurve1(CLK:=xProgCurve1, Q=>xDoIt);
   IF xyChart.xProgMode = FALSE THEN                              // If it's not already in programming mode
      xyChart.wsFocus := SVCurve1.wsCvName;                       // We need to inform the element, what's the curve that has the focus 
      IF iCurve1ProgType = 0 THEN
         xyChart.eProg := VisuEnumXYChartProgType.MODIFY;         // We inform the element to enter in programming mode for exixting curve modification
      ELSE   
         xyChart.eProg := VisuEnumXYChartProgType.NEW_CURVE;      // We inform the element to enter in programming mode for a new curve modify
      END_IF
      udiCycleCounter  := VisuSync.udiCycleCounter;               // We save the actual cycle counter 
      xDelayProgCurve1 := TRUE;
   END_IF
END_IF

// We wait some cycles before to act in programming mode,
// to give to the element the time to activate the programming mode
IF xDelayProgCurve1 THEN
   IF xyChart.xProgMode THEN                                            // Command has been executed
      xDelayProgCurve1       := FALSE;
      Curve1.ePointStyle     := VisuEnumXYChartPointStyle.DOT;          // We set the visualization of the line using also dot  
      xyChart.eFocusDisplay  := VisuEnumXYChartFocusType.FOC_REV_COL;   // We show the axis that has the focus, with reverse colors on numbers
      xyChart.diCursorColorM := VisuElemXYChart.COLOR.Red;              // We change the color of the cursor
	ELSE
      IF ABS(VisuSync.udiCycleCounter - udiCycleCounter) > 100 THEN
         xDelayProgCurve1 := FALSE;                                     // Something went wrong 
      END_IF
   END_IF
END_IF


//------------------------------------------------------------------
// We stop the programming
rTrigProgOff(CLK:=xProgOff, Q=>xDoIt);
IF xDoIt THEN
   xProgOff := FALSE;
   rTrigProgOff(CLK:=xProgOff, Q=>xDoIt);
   xyChart.eProg   := VisuEnumXYChartProgType.NO;    // We inform the element to stop the programming mode for a new curve modify 
   udiCycleCounter := VisuSync.udiCycleCounter;      // We save the actual cycle counter 
   xDelayProgOff   := TRUE;
END_IF

// We wait some cycles before to exit from programming mode,
// to give to the element the time to update the visualization
IF xDelayProgOff THEN
   IF NOT xyChart.xProgMode THEN                                  // Command has been executed
      xDelayProgOff          := FALSE;
      Curve1.ePointStyle     := SVCurve1.ePointStyle;             // We change it to the original one
      xyChart.wsFocus        := SVCurve1.wsCvName;                // We set the focus as default on curve1 
      xyChart.eFocusDisplay  := SVxyChart.eFocusDisplay;          // We change it to the original one
      xyChart.diCursorColorM := SVxyChart.diCursorColorM;         // We change it to the original one    
	ELSE
      IF ABS(VisuSync.udiCycleCounter - udiCycleCounter) > 100 THEN
         xDelayProgOff := FALSE;                                  // Something went wrong 
      END_IF
   END_IF
END_IF


//------------------------------------------------------------------
// We save the curve 
rTrigSave(CLK:=xProgSave, Q=>xDoIt);
IF xDoIt THEN
   xProgSave := FALSE;
   rTrigSave(CLK:=xProgSave, Q=>xDoIt);
   xyChart.eCommand := VisuEnumXYChartCommands.PRG_SAVE;          // We inform the element to save the curvestop the programming mode for a new curve modify
   udiCycleCounter := VisuSync.udiCycleCounter;                   // We save the actual cycle counter 
   xDelayProgSave := TRUE;
END_IF

// We wait some cycles,
// to give to the element the time to save all the data
IF xDelayProgSave THEN
   IF xyChart.eCommand = VisuEnumXYChartCommands.NO THEN   // Command has been executed
      xDelayProgSave := FALSE;
      xProgOff := TRUE;                                    // We will do the same operations like programming off 
	ELSE
      IF ABS(VisuSync.udiCycleCounter - udiCycleCounter) > 100 THEN
         xDelayProgSave := FALSE;                          // Something went wrong 
      END_IF
   END_IF
END_IF


//------------------------------------------------------------------
// Undo single point 
rTrigUndoS(CLK:=xProgUndoS, Q=>xDoIt);
IF xDoIt THEN
   xProgUndoS := FALSE;
   rTrigUndoS(CLK:=xProgUndoS, Q=>xDoIt);
   xyChart.eCommand := VisuEnumXYChartCommands.PRG_UNDO;
END_IF


//------------------------------------------------------------------
// Undo all 
rTrigUndo(CLK:=xProgUndo, Q=>xDoIt);
IF xDoIt THEN
   xProgUndo := FALSE;
   rTrigUndo(CLK:=xProgUndo, Q=>xDoIt);
   xyChart.eCommand := VisuEnumXYChartCommands.PRG_UNDO_ALL;
END_IF


//------------------------------------------------------------------
// Set original curve 
rTrigOrig(CLK:=xSetOrigCurve, Q=>xDoIt);
IF xDoIt THEN
   xSetOrigCurve := FALSE;
   rTrigOrig(CLK:=xSetOrigCurve, Q=>xDoIt);

   // We set all the data as the original   
   xyChart := SVxyChart;
   AxisX   := SVAxisX;
   AxisY1  := SVAxisY1;
   Curve1  := SVCurve1;

   // We limit the use of the array
   Curve1.diIndexMin := 1 ;        
   Curve1.diIndexMax := 10 ;
   
   FctSetDefaultDataCurve();  // Set default data for curves   
END_IF


//------------------------------------------------------------------
// On line situation 
sProgClient := VisuElemXYChart.VisuFctGetClientName(xyChart.eClientProg);     // On which client programming is active
xProgMode := xyChart.xProgMode;                                               // Element is in programming mode
xChangePending := xyChart.xChangePending;                                     // Change is pending

END_PROGRAM

// Device/Application/VISU
FUNCTION_BLOCK VISU
VAR_INPUT
END_VAR
VAR_OUTPUT
END_VAR
VAR
END_VAR

// 	TEMP_DEV_STATUS       : DWORD;
// 	HUM_DEV_STATUS        : DWORD;
// 	FAN_DEVICE_STATUS     : DWORD;
// 	HEATING_DEVICE_STATUS : DWORD;
// 	COOLING_DEVICE_STATUS : DWORD;

END_FUNCTION_BLOCK

// Device/Application/Overlap/Overlap
PROGRAM Overlap

VAR_INPUT
	xyChart: VisuStructXYChart;         // Variable for element configuration
   
	AxisX: VisuStructXYChartAxis;       // Variable for dynamic X axis configuration
	AxisY1 : VisuStructXYChartAxis;     // Variable for dynamic Y1 axis configuration
   
   Curve : VisuStructXYChartCurve;     // Variable for dynamic curve configuration

   // Arrays of data used for curves   
   DataX : ARRAY [1..200] OF REAL ;
   DataY : ARRAY [1..200] OF REAL ;
   
   iCurveHeapSize : INT := 4;    // Heap size
   iNumCurve : INT;              // Curves to display
   
	xStart : BOOL;          // Execution start/stop
   sText : STRING;         // text for button
   rOffset : REAL;         // Curve offset
   xShowTrace : BOOL;      // Show the tracing 
   xNotVisMsg : BOOL := TRUE;
   xChangeZoom : BOOL;
END_VAR

VAR
   xFirst : BOOL := TRUE;        // First entry in the loop
   xDoIt : BOOL;
   ePendingCmd : ENUM_CMD_PENDING := ENUM_CMD_PENDING.NO_CMD;         // There's a command pending
   rTrigStart :  R_TRIG;         // Trigger to detect start execution
   fTrigTimer :  F_TRIG;         // Trigger to detect square wave timer
   rTrigZoom :   R_TRIG;         // Trigger to detect zoom changing
   iCalc : INT;                  // Value for calculation
   iLoop : INT;                  // Loops already executed
   ix : INT;                     // General index 
   timer : TP ;                  // Timer for curve growing effect
	sampleTime : TIME := T#40MS;  // Timer value for curve growing effect
   xTimerEnd : BOOL;             // Bool for timer elapsing   
	rXValue : REAL;               // X value 
	rYValue : REAL;               // Y value 
   udiCycleCounter : UDINT;      // System cycle counter 
   udiCycleWait : UDINT;         // How many cycle to wait 
   tDelay : TON;
   xDelay : BOOL;
   xDelayEnd : BOOL;
   iActualZoom : INT;
END_VAR

(**********************************************************************************************
   The scope of this application is to show how to use XYChart element in overlapping mode.
   It simply generates a curve and when the curve arrives at a certain point,
   it informs the element to push it in the heap.
   The next curve is generated with an offset on X and Y, to have the possibility to see the 
   difference with the previous one.
   When we reach the maximum number of curves to display, we will clean all and start again
***********************************************************************************************)


//------------------------------------------------------------------
// Initial settings
IF xFirst THEN
   Curve.iCurveHeapSize := iCurveHeapSize;                  // We will maintain 4 curves in the heap
   Curve.eOverlap := VisuEnumXYChartCvOverlapType.OVERLAP;  // We will work in overlapping mode 
   Curve.diIndexMin := 1;                                   // We set the initial indexes to use
   Curve.diIndexMax := 1;
   iNumCurve := Curve.iCurveHeapSize;                       // We will display as many curves as the heap size
   xNotVisMsg := TRUE;
END_IF

//------------------------------------------------------------------
// We change the text of the button
IF xStart THEN
   sText := 'Stop drawing';
ELSE   
   sText := 'Start drawing';
END_IF   

//------------------------------------------------------------------
// We enable/disable the tracking of the curve drawing using level lines
xDoIt := FALSE;
IF xShowTrace THEN
   xDoIt := TRUE;
END_IF   
AxisX.aLevelLine[1].xEnable  := xDoIt;
AxisY1.aLevelLine[1].xEnable := xDoIt;

//------------------------------------------------------------------
// Detect the zoom cahnging 
rTrigZoom(CLK:=xChangeZoom, Q=>xDoIt);
IF xDoIt THEN
   xChangeZoom := xDoIt := FALSE;
   IF iActualZoom = 0 THEN
      iActualZoom := 1;
      AxisX.rMin := -5;
      AxisX.rMax := 20;
      AxisY1.rMin := 0;
      AxisY1.rMax := 10;
   ELSE   
      iActualZoom := 0;
      AxisX.rMin := -2;
      AxisX.rMax := 15;
      AxisY1.rMin := -1;
      AxisY1.rMax := 5;
	END_IF
END_IF   
 
//------------------------------------------------------------------
// We start the curve drawing 
rTrigStart(CLK:=xStart, Q=>xDoIt);
IF xDoIt THEN
   xDoIt := FALSE;
   // We clean up the arrays
   FOR ix := 1 TO 200 BY 1 DO
       DataX[ix] := 0.0;
       DataY[ix] := 0.0;
   END_FOR
   iCalc := 1;          // The initial calculation point of our curve
   iLoop := 0;          // No loop right now
   rOffset := 0.0;      // No curve offset right now
   
   // If we did a "start" and next a "stop", we can have some curves in the heap.
   // In this way we will remove them
   Curve.eCurveHeapCmd := VisuEnumXYChartCvHeapCmd.CLEAN;
   udiCycleCounter := VisuSync.udiCycleCounter;  // Save cycle counter 
   ePendingCmd := ENUM_CMD_PENDING.CLEAN;
   udiCycleWait := 10;                 // How many cycle to wait the command ending  
   xNotVisMsg := TRUE;
END_IF

//------------------------------------------------------------------
// Timer for data generation 
timer(IN:=xStart, PT:=sampleTime, Q=>xTimerEnd) ;
IF xTimerEnd = FALSE THEN
   timer(IN:=xTimerEnd, PT:=sampleTime, Q=>xTimerEnd) ;
END_IF ;
	
// Timer clock detection
fTrigTimer(CLK:=xTimerEnd, Q=>xDoIt) ;
IF xDoIt THEN
   xDoIt := FALSE;
   IF (ePendingCmd = ENUM_CMD_PENDING.NO_CMD) AND NOT xDelay THEN   // only if we don't have pending command
      
      // When arrive the tick of the clock
      // we do the curve calculation
      IF iCalc <= 126 THEN                            // If we are in the calculation limit
         FctGetXYValues(iCalc-1, rXValue, rYValue);   // Get new values  
         DataX[iCalc] := rXValue + rOffset;           // Store the value in the arrays
         DataY[iCalc] := rYValue + rOffset;
         Curve.diIndexMax := iCalc;                   // The last valid value in the array 
         iCalc := iCalc+1;                      
      ELSE                       // We have finish to calculate the curve
         xDelay := TRUE;         // Enable delay time to finish the display curve
		END_IF
      AxisX.aLevelLine[1].rValue  := DataX[Curve.diIndexMax];      // Update the position for curve tracking
      AxisY1.aLevelLine[1].rValue := DataY[Curve.diIndexMax];
   END_IF
END_IF

//------------------------------------------------------------------
// Test the delay time to finish the display curve 
tDelay(IN:=xDelay, PT:=T#2S, Q=>xDelayEnd);
IF xDelay THEN
   IF xDelayEnd THEN
      xDelay := FALSE;
      
      // We have finish to calculate the curve
      iCalc := 1;                            // Reset the calculation value
      iLoop := iLoop+1;                      // We are facing a new loop
      IF iLoop < iNumCurve THEN              // I've room again, update the curve !
         Curve.eCurveHeapCmd := VisuEnumXYChartCvHeapCmd.UPDATE;     // We update the curve
         ePendingCmd := ENUM_CMD_PENDING.UPDATE;  // Update pending
      ELSE                                   // Heap full
         iLoop := 0 ;                        // We will start with a neww loop
         Curve.eCurveHeapCmd := VisuEnumXYChartCvHeapCmd.CLEAN;     // We clean the heap   
         ePendingCmd := ENUM_CMD_PENDING.CLEAN;   // Clean 
         udiCycleWait := 50;                 // How many cycle to wait the command ending, to have time to see the last curve, before clean all 
         xNotVisMsg := FALSE;
      END_IF    
	END_IF
   udiCycleCounter := VisuSync.udiCycleCounter;  // save cycle counter 
END_IF

//------------------------------------------------------------------
// If there's a clean command pending, we wait some cycles
// to have the possibility to see the last curve
IF ePendingCmd = ENUM_CMD_PENDING.CLEAN THEN
   IF (ABS(VisuSync.udiCycleCounter - udiCycleCounter) > udiCycleWait) AND (Curve.eCurveHeapCmd = VisuEnumXYChartCvHeapCmd.NO) THEN
      iLoop := 0 ;                        // We will start with a neww loop
      rOffset := 0.0;                     // No curve offset
      ePendingCmd := ENUM_CMD_PENDING.NO_CMD;      
      xNotVisMsg := TRUE;
   END_IF
END_IF

//----------------------------------------------------------------------------------------
// If there's an update command pending, we simply wait the end of the command
IF ePendingCmd = ENUM_CMD_PENDING.UPDATE THEN
   IF Curve.eCurveHeapCmd = VisuEnumXYChartCvHeapCmd.NO THEN
      iCalc := 1;                         // Reset the calculation value
      rOffset := rOffset + 0.3;           // Next curve will have an offset
      Curve.diIndexMax := iCalc;          // Reset to init curve
      ePendingCmd := ENUM_CMD_PENDING.NO_CMD;      
      xNotVisMsg := TRUE;
   END_IF
END_IF

xFirst := FALSE;

END_PROGRAM

// Device/Application/LIMIT_CHECK
FUNCTION LIMIT_CHECK : BOOL
VAR_INPUT
	INPUT : REAL;
	UPPER_LIMIT : REAL;
	LOWER_LIMIT : REAL;
END_VAR
VAR
END_VAR


// Hysterese nicht vergessen 
IF INPUT >= UPPER_LIMIT OR INPUT <= LOWER_LIMIT THEN
	LIMIT_CHECK := TRUE;
ELSE
	LIMIT_CHECK := FALSE;
END_IF

END_FUNCTION

// Device/Application/READ_TRENDS
FUNCTION_BLOCK READ_TRENDS
VAR_INPUT
    xExecute : BOOL;
    sTrendName : STRING; (* Name of the Trend Recording *)
    tStartTime : DT;
    tEndTime : DT;
    iChannelIndex : INT := 0; 
END_VAR
VAR_IN_OUT
    stChartData : GRAPH_AXIS;
END_VAR
VAR_OUTPUT
    sLabels : STRING(2000); (* JSON array of labels *)
    xDone : BOOL;
    xBusy : BOOL;
    xError : BOOL;
    sError : STRING;
END_VAR
VAR
    step : INT := 0;
    i : DINT;
    
    // Fake data generation vars
    sTempLabel : STRING(20);
    dtCurrent : DT;
    iMaxLabels : INT := 20; 
END_VAR

CASE step OF
    0: (* Idle *)
        IF xExecute THEN
            xBusy := TRUE;
            xDone := FALSE;
            xError := FALSE;
            sError := '';
            step := 10;
        END_IF
        
    10: (* Start Read *)
        sLabels := '[';
        stChartData.diNumOfData := 100; (* Demo count *)
        
        (* Populate Data & Labels *)
        FOR i := 0 TO stChartData.diNumOfData - 1 DO
             // Simulate data
             stChartData.aData[i] := SIN(TO_REAL(i) * 0.1) * 10.0 + 20.0;
             
             // Construct Labels (limited subset)
             IF i < iMaxLabels THEN
                dtCurrent := tStartTime + TO_TIME(i * 60000); 
                sTempLabel := DT_TO_STRING(dtCurrent);
                sTempLabel := RIGHT(sTempLabel, 8); 
                
                IF i > 0 THEN
                    sLabels := CONCAT(sLabels, ', "');
                ELSE
                    sLabels := CONCAT(sLabels, '"');
                END_IF
                
                sLabels := CONCAT(sLabels, sTempLabel);
                sLabels := CONCAT(sLabels, '"');
             END_IF
        END_FOR
        
        sLabels := CONCAT(sLabels, ']');
        
        stChartData.sLabel := 'Trend Data';
        stChartData.sBorderColor := 'blue';
        stChartData.xFill := FALSE;
        
        step := 20;
        
    20: (* Done *)
        xDone := TRUE;
        xBusy := FALSE;
        IF NOT xExecute THEN
            step := 0;
        END_IF
        
END_CASE

END_FUNCTION_BLOCK

// Device/Application/DAY_TO_TIME
FUNCTION DAY_TO_TIME : TIME
VAR_INPUT
		IN : REAL;
END_VAR
VAR
END_VAR

DAY_TO_TIME := DWORD_TO_TIME(REAL_TO_DWORD(IN * 86400000.0));

END_FUNCTION

// Device/Application/Page
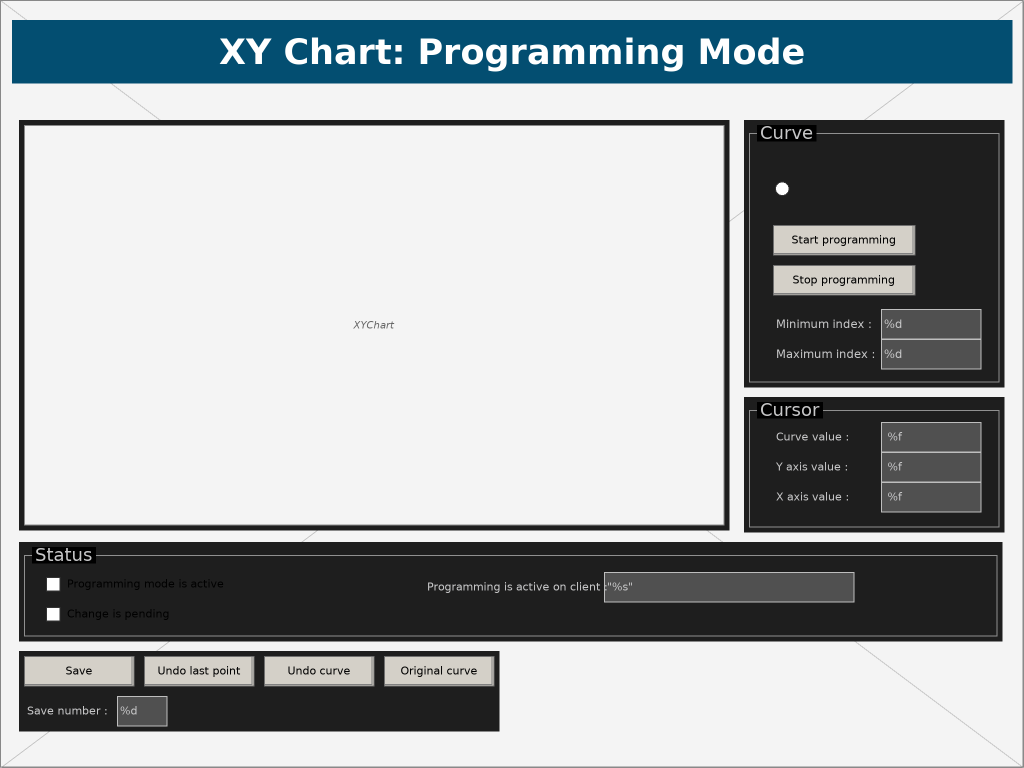
VISUALIZATION Page  // 1024x768
    Image (0,0 1024x768), image: ImagePool.background
    Rectangle (19,120 710x410)
    Rectangle (744,120 260x267)
    Rectangle (744,397 260x135)
    Rectangle (19,651 480x80)
    Rectangle (19,542 983x99)
    Button (384,656 110x30), "Original curve", input disabled if: prog.xyChart.xProgMode
        OnMouseClick:  ToggleVariable=Prog.xSetOrigCurve
    Button (24,656 110x30), "Save", input disabled if: not prog.xyChart.xProgMode
        OnMouseClick:  ToggleVariable=Prog.xProgSave
    Button (144,656 110x30), "Undo last point", input disabled if: not prog.xyChart.xProgMode
        OnMouseClick:  ToggleVariable=Prog.xProgUndoS
    Button (264,656 110x30), "Undo curve", input disabled if: not prog.xyChart.xProgMode
        OnMouseClick:  ToggleVariable=Prog.xProgUndo
    XYChart (24,125 700x400)
    GroupBox (749,125 250x257), "Curve"
        RadioButton (24,32 197x63), variable: Prog.iCurve1ProgType
            Areas[0]: Text=Modify the existing curve
            Areas[1]: Text=Create a new curve
        Button (24,100 142x30), "Start programming", input disabled if: prog.xyChart.xProgMode
            OnMouseClick:  ToggleVariable=Prog.xProgCurve1
        Button (24,140 142x30), "Stop programming", input disabled if: Not prog.xyChart.xProgMode
            OnMouseClick:  ToggleVariable=Prog.xProgOff
        Rectangle (132,184 100x30), "%d", text variable: Prog.Curve1.diIndexMin
            OnMouseClick: write the text variable via Default, min 1, max 98
        Rectangle (132,214 100x30), "%d", text variable: Prog.Curve1.diIndexMax
            OnMouseClick: write the text variable via Default, min 2, max 100
        Label (24,184 100x30), "Minimum index :"
        Label (24,214 100x30), "Maximum index :"
    GroupBox (749,402 250x125), "Cursor"
        Label (24,80 100x30), "X axis value :"
        Label (24,50 100x30), "Y axis value :"
        Label (24,20 100x30), "Curve value :"
        Rectangle (132,20 100x30), "%f", text variable: Prog.Curve1.rValueCursM
        Rectangle (132,50 100x30), "%f", text variable: Prog.AxisY1.rValueCursM
        Rectangle (132,80 100x30), "%f", text variable: Prog.AxisX.rValueCursM
    GroupBox (24,547 973x89), "Status"
        Checkbox (20,25 200x24), "Programming mode is active", variable: Prog.xProgMode, invisible if: FALSE, input disabled if: TRUE
        Checkbox (20,55 200x24), "Change is pending", variable: Prog.xChangePending, invisible if: FALSE, input disabled if: TRUE
        Rectangle (580,25 250x30), ""%s"", text variable: Prog.sProgClient
        Label (400,25 200x30), "Programming is active on client :"
    Rectangle (117,696 50x30), "%d", text variable: Prog.xyChart.udiPrgUpdateCtr
        OnMouseClick: write the text variable via Default, min 1, max 98
    Label (24,696 90x30), "Save number :"
    Rectangle (12,20 1000x63), "XY Chart: Programming Mode"
END_VISUALIZATION

// Device/Application/Visualization_1
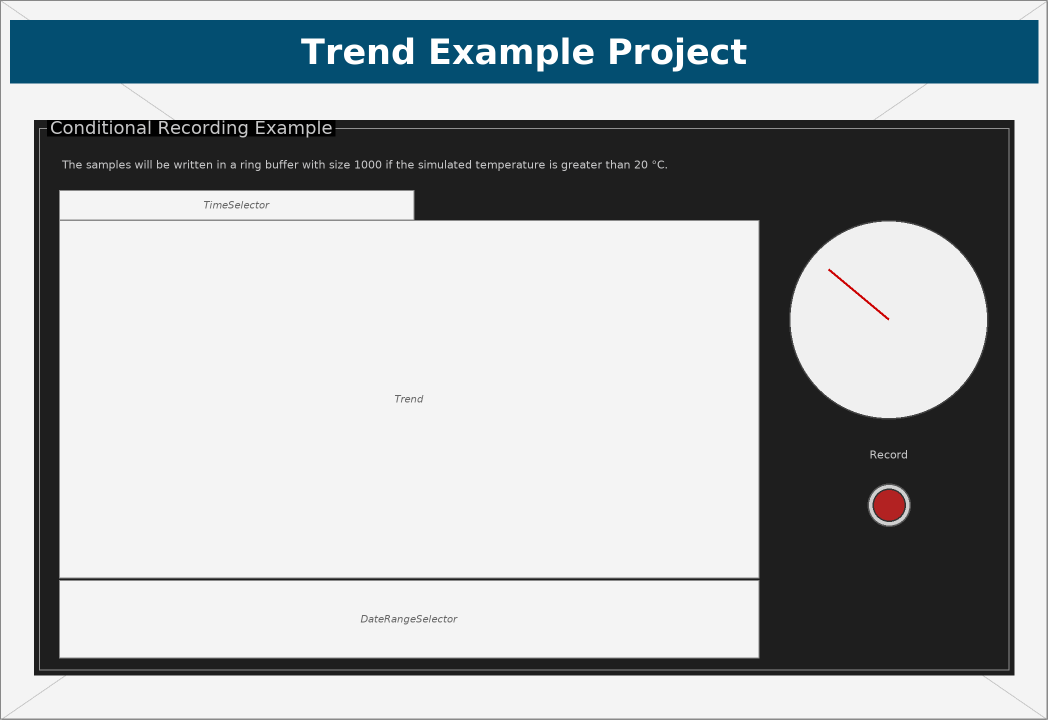
VISUALIZATION Visualization_1  // 1048x720
    Image (0,0 1048x720), image: ImagePool.background
    Rectangle (34,120 980x555)
    GroupBox (39,120 970x550), "Conditional Recording Example"
    Trend (59,220 700x358)
        p758368661: dd.MM.yyyy
        p2423372160: HH:mm:ss:ms
        p2833066001: Trend1
        p2059293862: GenElemInst_3
        p2541140726: GenElemInst_4
    DateRangeSelector (59,580 700x78)
        p758368661: dd.MM.yyyy
        p2423372160: HH:mm:ss:ms
        p1661464551: GenElemInst_1
    TimeSelector (59,190 355x30)
        p677259794: Zoom:
        p3737533738: GenElemInst_1
    Lamp1 (864,480 50x50), variable: PLC_PRG.xRecord, style: Lamp-Lamp1-Red
    Label (854,440 70x30), "Record"
    Label (59,150 600x30), "The samples will be written in a ring buffer with size 1000 if the simulated temperature is greater than 20 °C."
    Meter360 (789,220 199x199), value: PLC_PRG.rSignalToRecord1, style: Meter-Meter360-Yellow, scale format: %.1f, scale 10..30
        p518627256: Temperature in °C
    Rectangle (10,20 1028x63), "Trend Example Project"
END_VISUALIZATION

// Device/Application/Visualization
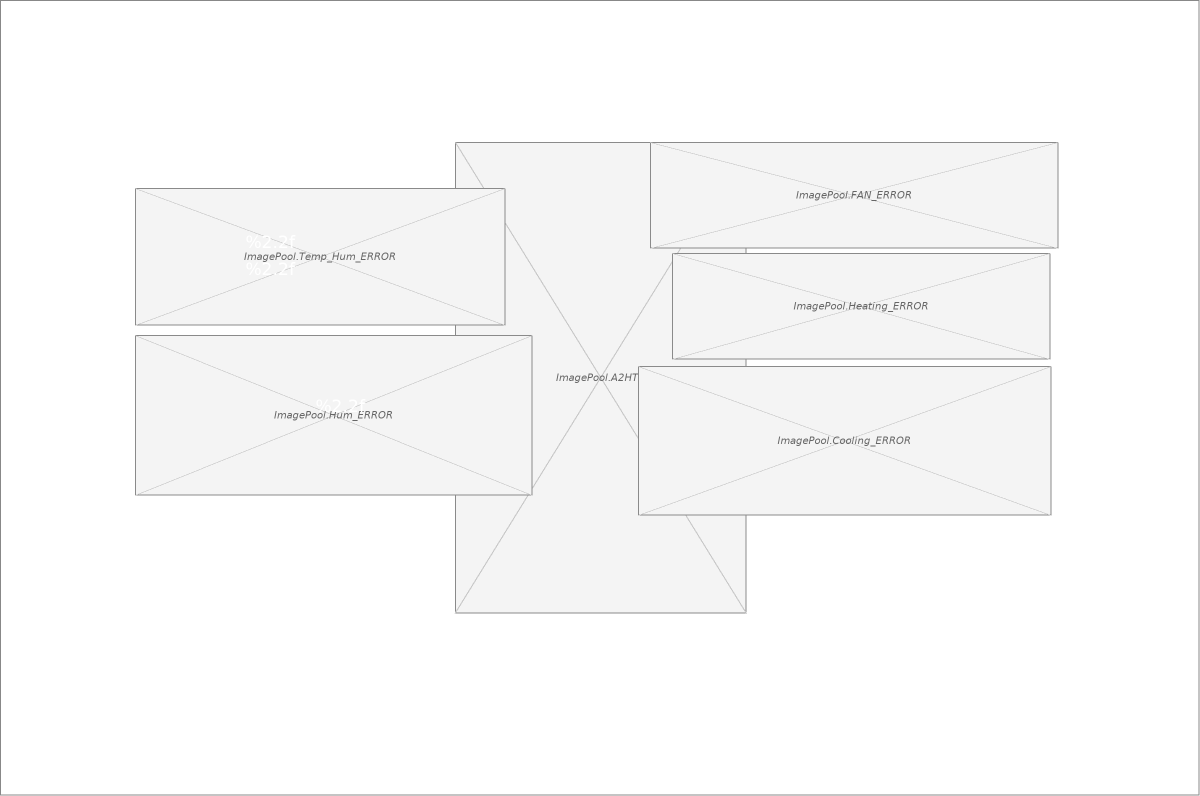
VISUALIZATION Visualization  // 1200x796, background image ImagePool.Hintergrund
    Image (455,142 291x471), image: ImagePool.A2HTC
    Image (135,188 370x137), image: ImagePool.Temp_Hum_OK
    Image (135,188 370x137), invisible if: NOT GVL.TEMP.STATUS.WARNING, image: ImagePool.Temp_Hum_WARN
    Image (135,188 370x137), invisible if: NOT GVL.TEMP.STATUS.ERROR, image: ImagePool.Temp_Hum_ERROR
    Rectangle (222,229 97x26), "%2.2f", text variable: GVL.TEMP.VALUE
    Rectangle (222,256 97x26), "%2.2f", text variable: GVL.TEMP.VALUE
    Image (135,335 397x160), image: ImagePool.HUM_OK
    Rectangle (297,390 97x26), text variable: GVL.TEMP.VALUE
    Image (135,335 397x160), invisible if: NOT GVL.HUM.STATUS.WARNING, image: ImagePool.Hum_WARN
    Image (135,335 397x160), invisible if: NOT GVL.HUM.STATUS.ERROR, image: ImagePool.Hum_ERROR
    Rectangle (292,393 97x26), "%2.2f", text variable: GVL.TEMP.VALUE
    Image (650,142 408x106), image: ImagePool.FAN_OK
    Image (672,253 378x106), image: ImagePool.Heating_OK
    Image (638,366 413x149), image: ImagePool.Cooling_OK
    Image (650,142 408x106), invisible if: NOT GVL.FAN.STATUS.WARNING, image: ImagePool.FAN_WARN
    Image (672,253 378x106), invisible if: NOT GVL.HEAT.STATUS.WARNING, image: ImagePool.Heating_WARN
    Image (638,366 413x149), invisible if: NOT GVL.COOLING.STATUS.WARNING, image: ImagePool.Cooling_WARN
    Image (650,142 408x106), invisible if: NOT GVL.FAN.STATUS.ERROR, image: ImagePool.FAN_ERROR
    Image (672,253 378x106), invisible if: NOT GVL.HEAT.STATUS.ERROR, image: ImagePool.Heating_ERROR
    Image (638,366 413x149), invisible if: NOT GVL.COOLING.STATUS.ERROR, image: ImagePool.Cooling_ERROR
END_VISUALIZATION

// Device/Application/Visualization_2
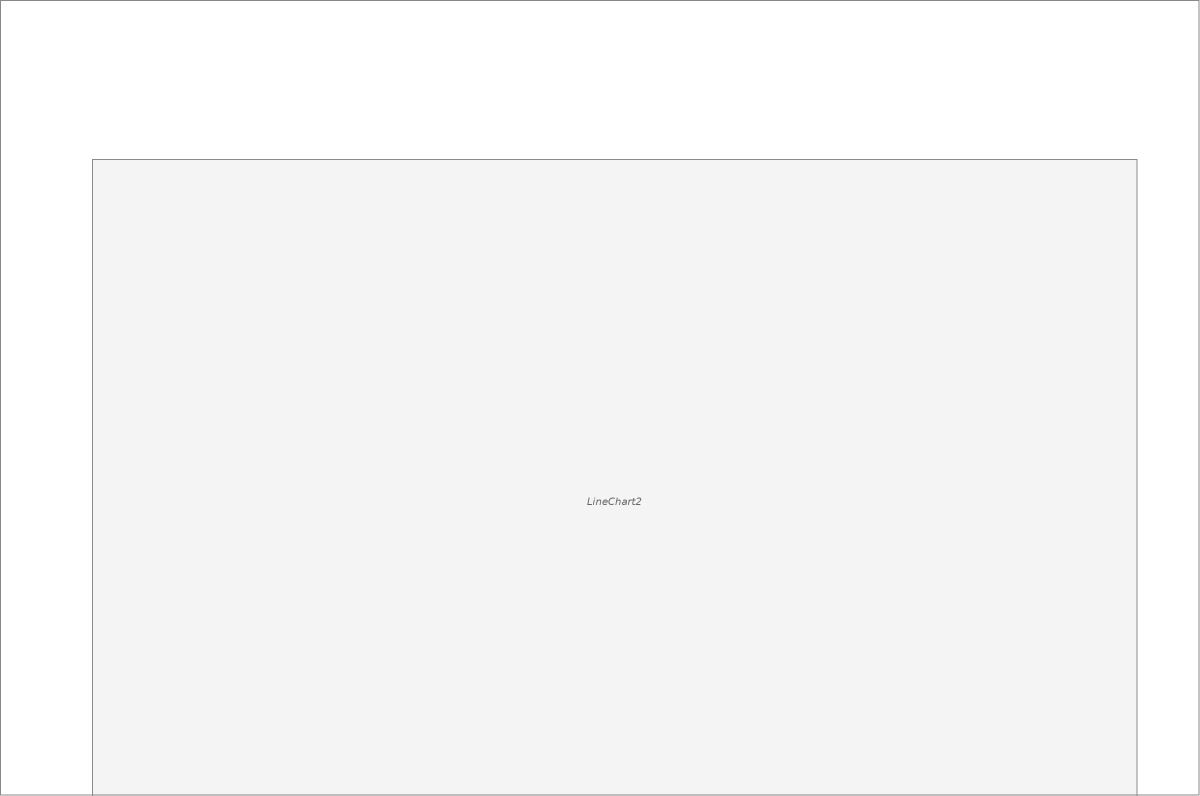
VISUALIZATION Visualization_2  // 1200x796
    LineChart2 (92,159 1045x685)
        p3734815120: TrendStorageAPI_TestProg.sLabelOne
        p4134829190: TrendStorageAPI_TestProg.ChartOne.aData
        p2520911902: TrendStorageAPI_TestProg.ChartOne.sBorderColor
        p2932080977: TrendStorageAPI_TestProg.ChartOne.xFill
        p2774779838: TrendStorageAPI_TestProg.ChartOne.diNumOfData
END_VISUALIZATION

// Device/Application/Visualizations/MinMaxTimestamps
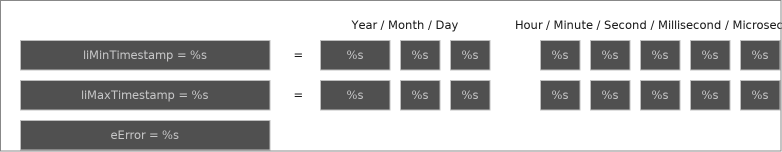
VISUALIZATION MinMaxTimestamps  // 782x152
    Rectangle (20,40 250x30), "liMinTimestamp = %s", text variable: TrendStorageAPI_TestProg.liMinTimestamp
        OnMouseClick: write the text variable via Default
    Rectangle (20,80 250x30), "liMaxTimestamp = %s", text variable: TrendStorageAPI_TestProg.liMaxTimestamp
        OnMouseClick: write the text variable via Default
    Rectangle (20,120 250x30), "eError = %s", text variable: TrendStorageAPI_TestProg.eError
    Rectangle (320,40 70x30), "%s", text variable: TrendStorageAPI_TestProg.timeDateMin.wYear
    Rectangle (400,40 40x30), "%s", text variable: TrendStorageAPI_TestProg.timeDateMin.wMonth
    Rectangle (450,40 40x30), "%s", text variable: TrendStorageAPI_TestProg.timeDateMin.wDay
    Rectangle (540,40 40x30), "%s", text variable: TrendStorageAPI_TestProg.timeDateMin.wHour
    Rectangle (640,40 40x30), "%s", text variable: TrendStorageAPI_TestProg.timeDateMin.wSecond
    Rectangle (690,40 40x30), "%s", text variable: TrendStorageAPI_TestProg.timeDateMin.wMilliseconds
    Rectangle (740,40 40x30), "%s", text variable: TrendStorageAPI_TestProg.uiMicrosecondsMin
    Rectangle (320,80 70x30), "%s", text variable: TrendStorageAPI_TestProg.timeDateMax.wYear
    Rectangle (400,80 40x30), "%s", text variable: TrendStorageAPI_TestProg.timeDateMax.wMonth
    Rectangle (450,80 40x30), "%s", text variable: TrendStorageAPI_TestProg.timeDateMax.wDay
    Rectangle (540,80 40x30), "%s", text variable: TrendStorageAPI_TestProg.timeDateMax.wHour
    Rectangle (640,80 40x30), "%s", text variable: TrendStorageAPI_TestProg.timeDateMax.wSecond
    Rectangle (690,80 40x30), "%s", text variable: TrendStorageAPI_TestProg.timeDateMax.wMilliseconds
    Rectangle (740,80 40x30), "%s", text variable: TrendStorageAPI_TestProg.uiMicrosecondsMax
    Label (280,40 37x30), "="
    Label (280,80 37x30), "="
    Label (320,10 170x30), "Year / Month / Day"
    Label (540,10 240x30), "Hour / Minute / Second / Millisecond / Microsecond"
    Rectangle (590,40 40x30), "%s", text variable: TrendStorageAPI_TestProg.timeDateMin.wMinute
    Rectangle (590,80 40x30), "%s", text variable: TrendStorageAPI_TestProg.timeDateMax.wMinute
END_VISUALIZATION

// Device/Application/Visualizations/ReadValues
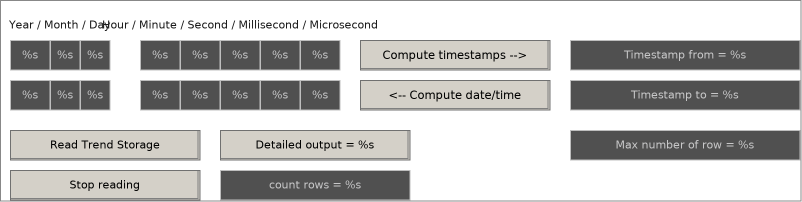
VISUALIZATION ReadValues  // 802x202
    Button (10,130 190x30), "Read Trend Storage"
        toggle TrendStorageAPI_TestProg.xDoReadTest2
    Rectangle (220,170 190x30), "count rows = %s", text variable: TrendStorageAPI_TestProg.instTrendStorageReaderConsumer.diTotalCountRows
    Rectangle (570,40 230x30), "Timestamp from = %s", text variable: TrendStorageAPI_TestProg.liTimstampFrom2
        OnMouseClick: write the text variable via Default
    Rectangle (570,80 230x30), "Timestamp to = %s", text variable: TrendStorageAPI_TestProg.liTimstampTo2
        OnMouseClick: write the text variable via Default
    Button (10,170 190x30), "Stop reading"
        toggle TrendStorageAPI_TestProg.xStopContinueReading
    Button (220,130 190x30), "Detailed output = %s", tooltip "If this option is activated a csv export will be simulated, i.e. the data will be dumped to the console in a format similar to csv", text variable: TrendStorageAPI_TestProg.instTrendStorageReaderConsumer.xDetailedOutput
        toggle TrendStorageAPI_TestProg.instTrendStorageReaderConsumer.xDetailedOutput
    Rectangle (10,40 40x30), "%s", text variable: TrendStorageAPI_TestProg.timeDateFrom2.wYear
        OnMouseClick: write the text variable via Default
    Rectangle (50,40 30x30), "%s", text variable: TrendStorageAPI_TestProg.timeDateFrom2.wMonth
        OnMouseClick: write the text variable via Default
    Rectangle (80,40 30x30), "%s", text variable: TrendStorageAPI_TestProg.timeDateFrom2.wDay
        OnMouseClick: write the text variable via Default
    Rectangle (140,40 40x30), "%s", text variable: TrendStorageAPI_TestProg.timeDateFrom2.wHour
        OnMouseClick: write the text variable via Default
    Rectangle (220,40 40x30), "%s", text variable: TrendStorageAPI_TestProg.timeDateFrom2.wSecond
        OnMouseClick: write the text variable via Default
    Rectangle (260,40 40x30), "%s", text variable: TrendStorageAPI_TestProg.timeDateFrom2.wMilliseconds
        OnMouseClick: write the text variable via Default
    Rectangle (300,40 40x30), "%s", text variable: TrendStorageAPI_TestProg.uiMicrosecondsFrom2
        OnMouseClick: write the text variable via Default
    Rectangle (10,80 40x30), "%s", text variable: TrendStorageAPI_TestProg.timeDateTo2.wYear
        OnMouseClick: write the text variable via Default
    Rectangle (50,80 30x30), "%s", text variable: TrendStorageAPI_TestProg.timeDateTo2.wMonth
        OnMouseClick: write the text variable via Default
    Rectangle (80,80 30x30), "%s", text variable: TrendStorageAPI_TestProg.timeDateTo2.wDay
        OnMouseClick: write the text variable via Default
    Rectangle (140,80 40x30), "%s", text variable: TrendStorageAPI_TestProg.timeDateTo2.wHour
        OnMouseClick: write the text variable via Default
    Rectangle (220,80 40x30), "%s", text variable: TrendStorageAPI_TestProg.timeDateTo2.wSecond
        OnMouseClick: write the text variable via Default
    Rectangle (260,80 40x30), "%s", text variable: TrendStorageAPI_TestProg.timeDateTo2.wMilliseconds
        OnMouseClick: write the text variable via Default
    Rectangle (300,80 40x30), "%s", text variable: TrendStorageAPI_TestProg.uiMicrosecondsTo2
        OnMouseClick: write the text variable via Default
    Label (10,10 100x30), "Year / Month / Day"
    Label (120,10 240x30), "Hour / Minute / Second / Millisecond / Microsecond"
    Rectangle (180,40 40x30), "%s", text variable: TrendStorageAPI_TestProg.timeDateFrom2.wMinute
        OnMouseClick: write the text variable via Default
    Rectangle (180,80 40x30), "%s", text variable: TrendStorageAPI_TestProg.timeDateTo2.wMinute
        OnMouseClick: write the text variable via Default
    Button (360,40 190x30), "Compute timestamps -->"
        toggle TrendStorageAPI_TestProg.xComputeTimestamps
    Button (360,80 190x30), "<-- Compute date/time"
        toggle TrendStorageAPI_TestProg.xComputeDateTime
    Rectangle (570,130 230x30), "Max number of row = %s", tooltip "This is the maximum number of rows a single read call can return. Decrease this value for slow devices.", text variable: TrendStorageReaderGlobals.g_iMaxCountRowsToRead
        OnMouseClick: write the text variable via Default
END_VISUALIZATION

// Device/Application/Visualizations/NewDataWritten
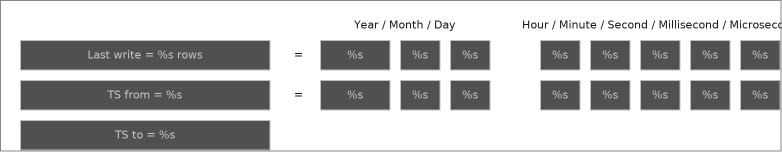
VISUALIZATION NewDataWritten  // 782x152
    Rectangle (20,40 250x30), "Last write = %s rows", text variable: TrendStorageAPI_TestProg.instTrendStorageWriterListener.m_iCountRows
    Rectangle (20,80 250x30), "TS from = %s", text variable: TrendStorageAPI_TestProg.instTrendStorageWriterListener.m_liFirstTimestamp
    Rectangle (20,120 250x30), "TS to = %s", text variable: TrendStorageAPI_TestProg.instTrendStorageWriterListener.m_liLastTimestamp
    Rectangle (320,40 70x30), "%s", text variable: TrendStorageAPI_TestProg.instTrendStorageWriterListener.m_timeDateMin.wYear
    Rectangle (400,40 40x30), "%s", text variable: TrendStorageAPI_TestProg.instTrendStorageWriterListener.m_timeDateMin.wMonth
    Rectangle (450,40 40x30), "%s", text variable: TrendStorageAPI_TestProg.instTrendStorageWriterListener.m_timeDateMin.wDay
    Rectangle (540,40 40x30), "%s", text variable: TrendStorageAPI_TestProg.instTrendStorageWriterListener.m_timeDateMin.wHour
    Rectangle (640,40 40x30), "%s", text variable: TrendStorageAPI_TestProg.instTrendStorageWriterListener.m_timeDateMin.wSecond
    Rectangle (690,40 40x30), "%s", text variable: TrendStorageAPI_TestProg.instTrendStorageWriterListener.m_timeDateMin.wMilliseconds
    Rectangle (740,40 40x30), "%s", text variable: TrendStorageAPI_TestProg.instTrendStorageWriterListener.m_uiMicrosecondsMin
    Rectangle (320,80 70x30), "%s", text variable: TrendStorageAPI_TestProg.instTrendStorageWriterListener.m_timeDateMax.wYear
    Rectangle (400,80 40x30), "%s", text variable: TrendStorageAPI_TestProg.instTrendStorageWriterListener.m_timeDateMax.wMonth
    Rectangle (450,80 40x30), "%s", text variable: TrendStorageAPI_TestProg.instTrendStorageWriterListener.m_timeDateMax.wDay
    Rectangle (540,80 40x30), "%s", text variable: TrendStorageAPI_TestProg.instTrendStorageWriterListener.m_timeDateMax.wHour
    Rectangle (640,80 40x30), "%s", text variable: TrendStorageAPI_TestProg.instTrendStorageWriterListener.m_timeDateMax.wSecond
    Rectangle (690,80 40x30), "%s", text variable: TrendStorageAPI_TestProg.instTrendStorageWriterListener.m_timeDateMax.wMilliseconds
    Rectangle (740,80 40x30), "%s", text variable: TrendStorageAPI_TestProg.instTrendStorageWriterListener.m_uiMicrosecondsMax
    Label (320,10 170x30), "Year / Month / Day"
    Label (540,10 240x30), "Hour / Minute / Second / Millisecond / Microsecond"
    Rectangle (590,40 40x30), "%s", text variable: TrendStorageAPI_TestProg.instTrendStorageWriterListener.m_timeDateMin.wMinute
    Rectangle (590,80 40x30), "%s", text variable: TrendStorageAPI_TestProg.instTrendStorageWriterListener.m_timeDateMax.wMinute
    Label (280,40 37x30), "="
    Label (280,80 37x30), "="
END_VISUALIZATION

(* text list TextList (id | default)
  cv1 | Curve 1
  posx | X
  posy | Y
  0 | 
  cv2 | Curve 2
   |  *)
